# EPICS autosave request: trunk/mcaApp/Db/RontecXFlash_settings.req
$(P)$(R)ReadTemperature.SCAN
$(P)$(R)SetMode
